Xinje XDPPro project, PLC1: XD5E-60T10 (software 3.5.3 2018-11-19)

PROGRAM Ladder

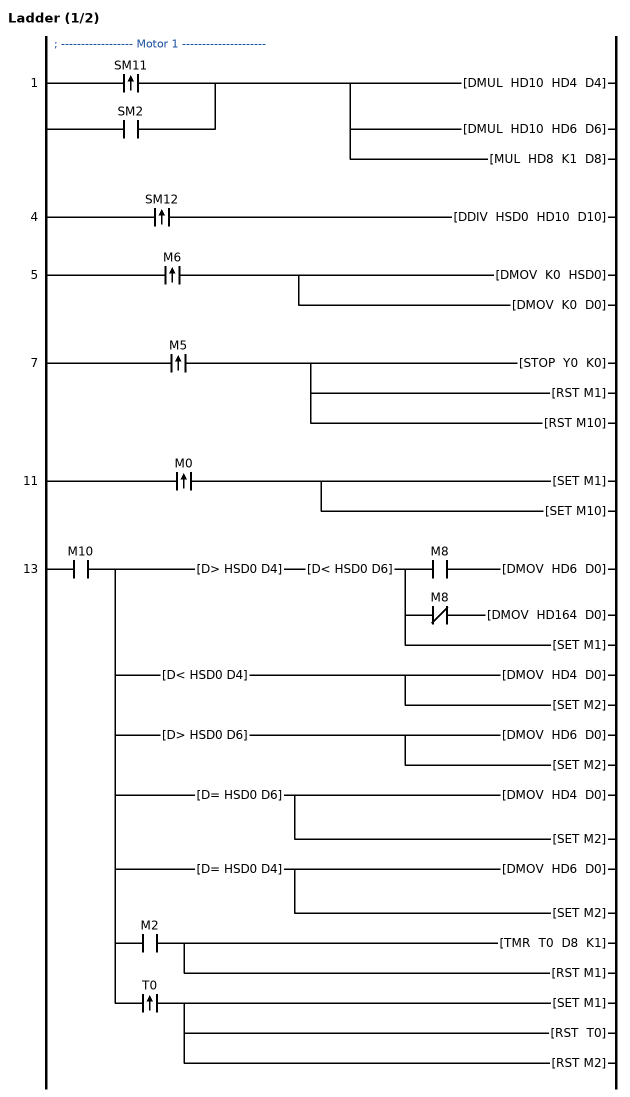
; ------------------ Motor 1 ---------------------
LDP    SM11
OR     SM2
DMUL   HD10 HD4 D4
DMUL   HD10 HD6 D6
MUL    HD8 K1 D8
LDP    SM12
DDIV   HSD0 HD10 D10
LDP    M6
DMOV   K0 HSD0
DMOV   K0 D0
LDP    M5
STOP   Y0 K0
RST    M1
RST    M10
LDP    M0
SET    M1
SET    M10
LD     M10
MPS
DAND>  HSD0 D4
DAND<  HSD0 D6
MPS
AND    M8
DMOV   HD6 D0
MRD
ANI    M8
DMOV   HD164 D0
MPP
SET    M1
MRD
DAND<  HSD0 D4
DMOV   HD4 D0
SET    M2
MRD
DAND>  HSD0 D6
DMOV   HD6 D0
SET    M2
MRD
DAND=  HSD0 D6
DMOV   HD4 D0
SET    M2
MRD
DAND=  HSD0 D4
DMOV   HD6 D0
SET    M2
MRD
AND    M2
TMR    T0 D8 K1
RST    M1
MPP
ANDP   T0
SET    M1
RST    T0
RST    M2

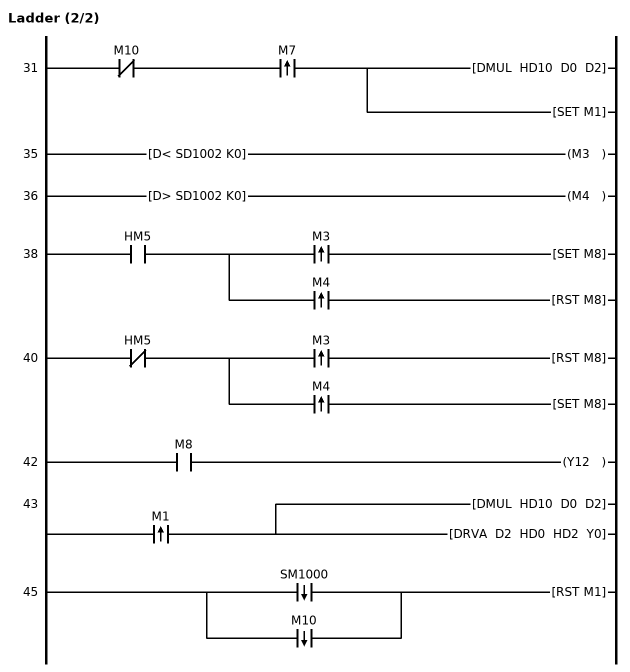
LDI    M10
ANDP   M7
DMUL   HD10 D0 D2
SET    M1
DLD<   SD1002 K0
OUT    M3
DLD>   SD1002 K0
OUT    M4
LD     HM5
MPS
ANDP   M3
SET    M8
MPP
ANDP   M4
RST    M8
LDI    HM5
MPS
ANDP   M3
RST    M8
MPP
ANDP   M4
SET    M8
LD     M8
OUT    Y12
LDP    M1
DMUL   HD10 D0 D2
DRVA   D2 HD0 HD2 Y0
LDF    SM1000
ORF    M10
RST    M1